Staubli VAL3: PULSE.dtx

public string sItems[2]
string sMessage
bool bExecute[3]
public string sItemsCycle
